FUNCTION "SCREEN 9 = FAULTS" : Void   // FC23, LAD
{ S7_Optimized_Access := 'TRUE' }
VERSION : 0.1
BEGIN
END_FUNCTION

FUNCTION "SCREEN 8 = ROBOT UR CONTROL" : Void   // FC24, LAD
{ S7_Optimized_Access := 'TRUE' }
VERSION : 0.1
BEGIN
END_FUNCTION

FUNCTION "SCREEN 10 = WARNINGS" : Void   // FC25, LAD
{ S7_Optimized_Access := 'TRUE' }
VERSION : 0.1
BEGIN
END_FUNCTION

FUNCTION "SCREEN 5 = SAFETY" : Void   // FC27, LAD
{ S7_Optimized_Access := 'TRUE' }
VERSION : 0.1
BEGIN
END_FUNCTION

FUNCTION "SCREEN 4 = RECIPE EDIT" : Void   // FC28, LAD
{ S7_Optimized_Access := 'TRUE' }
VERSION : 0.1
BEGIN
END_FUNCTION

FUNCTION "SCREEN 3 = RECIPE SELECT" : Void   // FC29, LAD
{ S7_Optimized_Access := 'TRUE' }
VERSION : 0.1
BEGIN
END_FUNCTION

FUNCTION "SCREEN 1 = MAIN" : Void   // FC30, LAD
{ S7_Optimized_Access := 'TRUE' }
VERSION : 0.1
BEGIN
END_FUNCTION

FUNCTION "SCREEN 6 = VISION CONTROL" : Void   // FC34, LAD
{ S7_Optimized_Access := 'TRUE' }
VERSION : 0.1
BEGIN
END_FUNCTION

// folder: UTILITIES OR DEVICES/UR

FUNCTION "UR CONTROL" : Void   // FC26, LAD
{ S7_Optimized_Access := 'TRUE' }
VERSION : 0.1
BEGIN
END_FUNCTION

FUNCTION "UR MANUAL SWITCH CASE" : Void   // FC33, LAD
{ S7_Optimized_Access := 'TRUE' }
VERSION : 0.1
BEGIN
END_FUNCTION

FUNCTION "UR PERMISSIVES" : Void   // FC35, LAD
{ S7_Optimized_Access := 'TRUE' }
VERSION : 0.1
BEGIN
END_FUNCTION